{attribute 'GeneratedUsingTerminal: EL9290--0000'}
{attribute addProperty BoxType "EL9290--0000"}
{attribute addProperty Description "EL9290 Power Supplier (Fuse)"}
{attribute addProperty Physics "KK"}
{attribute addProperty Id "EL9290"}
{attribute addProperty CRC "1533360857"}
{attribute addProperty Size "0"}
TYPE EL9290_5B653AD9 EXTENDS EtcSlaveTerminalBase_947E5A46 :
STRUCT
END_STRUCT
END_TYPE

(* stored: Version 1.2.0.0, ProductVersion 3.1.4024.11
   DUT EL9290_5B653AD9: Id {1f657ed3-994f-43f0-8613-e51bd50cd156} *)
